// TIA Portal V19 export
ORGANIZATION_BLOCK "RT_Info_Cyclic"   // OB30, LAD, CyclicInterrupt
{ S7_Optimized_Access := 'TRUE' }
// stored: SetENOAutomatically false
   VAR_INPUT
      Initial_Call : Bool;   // Initial call of this OB
      Event_Count : Int;   // Events discarded
   END_VAR
   VAR CONSTANT
      constRunSoloState : Int := 37;
      constRunRedundant : Int := 40;
   END_VAR
   VAR_TEMP   // added for the SCL form of the ladder/FBD networks
      _w1 : Bool;
      _w2 : Bool;
      _w3 : Bool;
      _w4 : Bool;
   END_VAR
BEGIN

REGION Network 1: RT_Info for specific OB
   // Used to find the specific runtime of an OB, change the OB number and see the INFO.
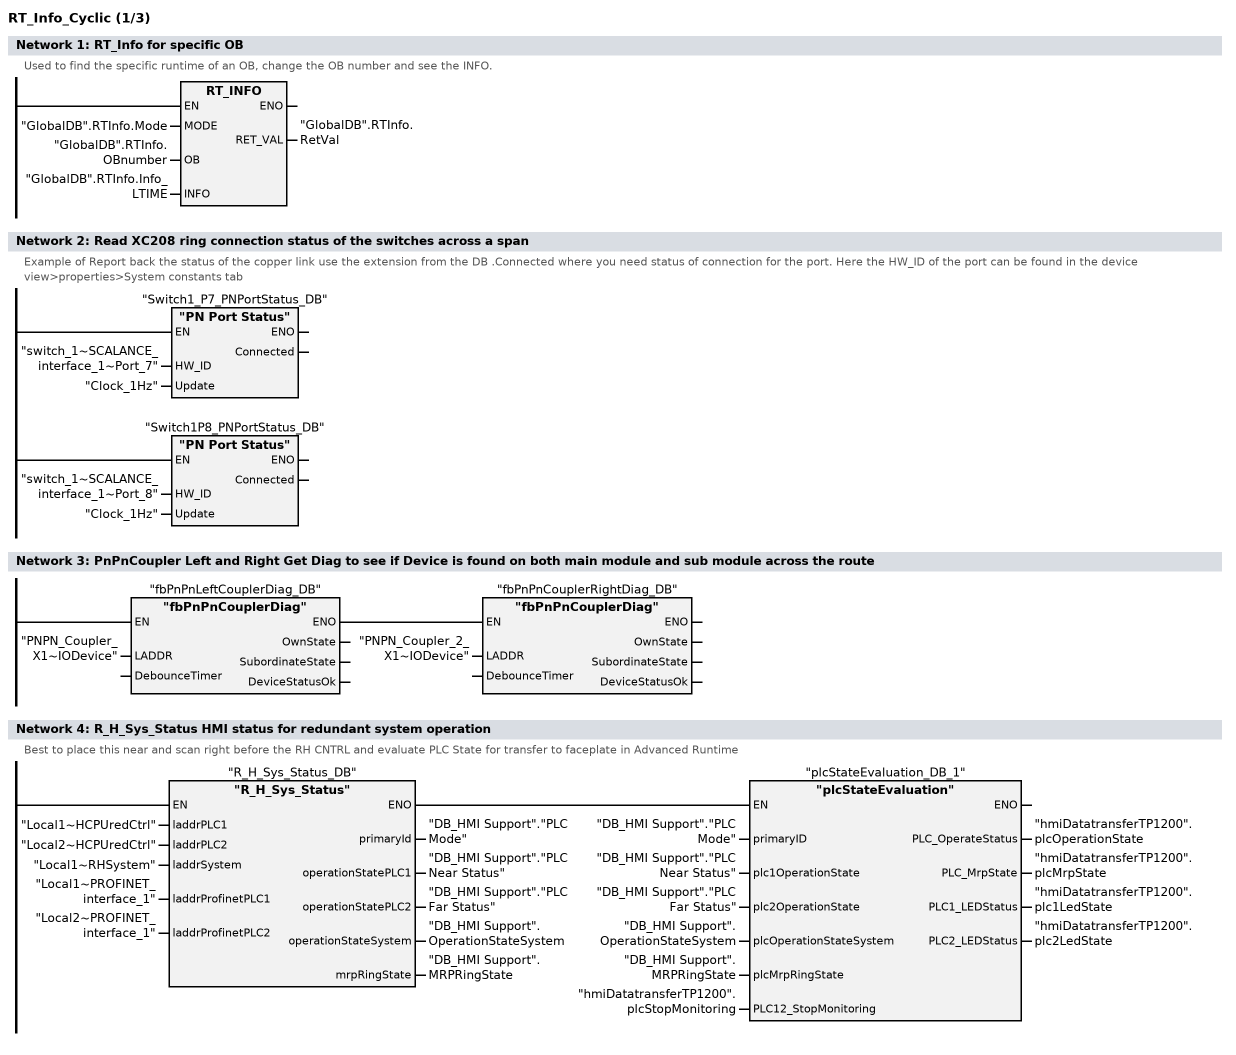
   RUNG wire#powerrail
      RT_INFO(MODE := "GlobalDB".RTInfo.Mode, OB := "GlobalDB".RTInfo.OBnumber, INFO := "GlobalDB".RTInfo.Info_LTIME, Ret_Val => "GlobalDB".RTInfo.RetVal)
   END_RUNG
   // the same network as SCL:
   "GlobalDB".RTInfo.RetVal := RT_INFO(MODE := "GlobalDB".RTInfo.Mode,
                           OB := "GlobalDB".RTInfo.OBnumber,
                           INFO := "GlobalDB".RTInfo.Info_LTIME);
END_REGION

REGION Network 2: Read XC208 ring connection status of the switches across a span
   // Example of Report back the status of the copper link use the extension from the DB .Connected where you need status of connection for the port. Here the HW_ID of the port can be found in the device view>properties>System constants tab
   RUNG wire#powerrail
      "Switch1_P7_PNPortStatus_DB"(HW_ID := "switch_1~SCALANCE_interface_1~Port_7", Update := "Clock_1Hz", Connected =>)
   END_RUNG
   RUNG wire#powerrail
      "Switch1P8_PNPortStatus_DB"(HW_ID := "switch_1~SCALANCE_interface_1~Port_8", Update := "Clock_1Hz", Connected =>)
   END_RUNG
   // the same network as SCL:
   "Switch1_P7_PNPortStatus_DB"(HW_ID := "switch_1~SCALANCE_interface_1~Port_7", Update := "Clock_1Hz");   // "PN Port Status"
   "Switch1P8_PNPortStatus_DB"(HW_ID := "switch_1~SCALANCE_interface_1~Port_8", Update := "Clock_1Hz");   // "PN Port Status"
END_REGION

REGION Network 3: PnPnCoupler Left and Right Get Diag to see if Device is found on both main module and sub module across the route
   RUNG wire#powerrail
      "fbPnPnLeftCouplerDiag_DB"(LADDR := "PNPN_Coupler_X1~IODevice", DebounceTimer :=, OwnState =>, SubordinateState =>, DeviceStatusOk =>)
      "fbPnPnCouplerRightDiag_DB"(LADDR := "PNPN_Coupler_2_X1~IODevice", DebounceTimer :=, OwnState =>, SubordinateState =>, DeviceStatusOk =>)
   END_RUNG
   // the same network as SCL:
   "fbPnPnLeftCouplerDiag_DB"(LADDR := "PNPN_Coupler_X1~IODevice", ENO => #_w1);   // "fbPnPnCouplerDiag"
   IF #_w1 THEN
       "fbPnPnCouplerRightDiag_DB"(LADDR := "PNPN_Coupler_2_X1~IODevice");   // "fbPnPnCouplerDiag"
   END_IF;
END_REGION

REGION Network 4: R_H_Sys_Status HMI status for redundant system operation
   // Best to place this near and scan right before the RH CNTRL and evaluate PLC State for transfer to faceplate in Advanced Runtime
   RUNG wire#powerrail
      "R_H_Sys_Status_DB"(laddrPLC1 := "Local1~HCPUredCtrl", laddrPLC2 := "Local2~HCPUredCtrl", laddrSystem := "Local1~RHSystem", laddrProfinetPLC1 := "Local1~PROFINET_interface_1", laddrProfinetPLC2 := "Local2~PROFINET_interface_1", primaryId => "DB_HMI Support"."PLC Mode", operationStatePLC1 => "DB_HMI Support"."PLC Near Status", operationStatePLC2 => "DB_HMI Support"."PLC Far Status", operationStateSystem => "DB_HMI Support".OperationStateSystem, mrpRingState => "DB_HMI Support".MRPRingState)
      "plcStateEvaluation_DB_1"(primaryID := "DB_HMI Support"."PLC Mode", plc1OperationState := "DB_HMI Support"."PLC Near Status", plc2OperationState := "DB_HMI Support"."PLC Far Status", plcOperationStateSystem := "DB_HMI Support".OperationStateSystem, plcMrpRingState := "DB_HMI Support".MRPRingState, PLC12_StopMonitoring := "hmiDatatransferTP1200".plcStopMonitoring, PLC_OperateStatus => "hmiDatatransferTP1200".plcOperationState, PLC_MrpState => "hmiDatatransferTP1200".plcMrpState, PLC1_LEDStatus => "hmiDatatransferTP1200".plc1LedState, PLC2_LEDStatus => "hmiDatatransferTP1200".plc2LedState)
   END_RUNG
   // the same network as SCL:
   "R_H_Sys_Status_DB"(laddrPLC1 := "Local1~HCPUredCtrl",   // "R_H_Sys_Status"
                       laddrPLC2 := "Local2~HCPUredCtrl",
                       laddrSystem := "Local1~RHSystem",
                       laddrProfinetPLC1 := "Local1~PROFINET_interface_1",
                       laddrProfinetPLC2 := "Local2~PROFINET_interface_1",
                       primaryId => "DB_HMI Support"."PLC Mode",
                       operationStatePLC1 => "DB_HMI Support"."PLC Near Status",
                       operationStatePLC2 => "DB_HMI Support"."PLC Far Status",
                       operationStateSystem => "DB_HMI Support".OperationStateSystem,
                       mrpRingState => "DB_HMI Support".MRPRingState,
                       ENO => #_w1);
   IF #_w1 THEN
       "plcStateEvaluation_DB_1"(primaryID := "DB_HMI Support"."PLC Mode",   // "plcStateEvaluation"
                               plc1OperationState := "DB_HMI Support"."PLC Near Status",
                               plc2OperationState := "DB_HMI Support"."PLC Far Status",
                               plcOperationStateSystem := "DB_HMI Support".OperationStateSystem,
                               plcMrpRingState := "DB_HMI Support".MRPRingState,
                               PLC12_StopMonitoring := "hmiDatatransferTP1200".plcStopMonitoring,
                               PLC_OperateStatus => "hmiDatatransferTP1200".plcOperationState,
                               PLC_MrpState => "hmiDatatransferTP1200".plcMrpState,
                               PLC1_LEDStatus => "hmiDatatransferTP1200".plc1LedState,
                               PLC2_LEDStatus => "hmiDatatransferTP1200".plc2LedState);
   END_IF;
END_REGION

REGION Network 5: Trigger primary stop RH_CNTRL
   // Self Latching Sequence using FullSwap Sequence tag, independent function with REQ tag
   // Used to trigger Primary Stop based on input from stop primary and full swap boolean tag;
   //  positive edge triggered instruction RH_CTRL below.
   // This network uses a Primary stop request, and evaluates if the RH_CTRL is busy before 
   // changing the mode or moving on to the next step.
   // The Retry_Busy tag is used to record if a Busy bit was in place while being triggered to prevent moving
   //  mode during middle of RH_CTRL operation.
   // 
   // Modes:
   // 3: Disable execution of the SYNCUP
   // 4: Re-enable execution of the SYNCUP
   // 7: Request SYNCUP system state 
   // 8: Request STOP of the primary CPU
   // 9: Request STOP of the backup CPU
   // 
   // Use mode 8 to stop the primary PLC, then use Mode 7 to Synch the primary and backup.
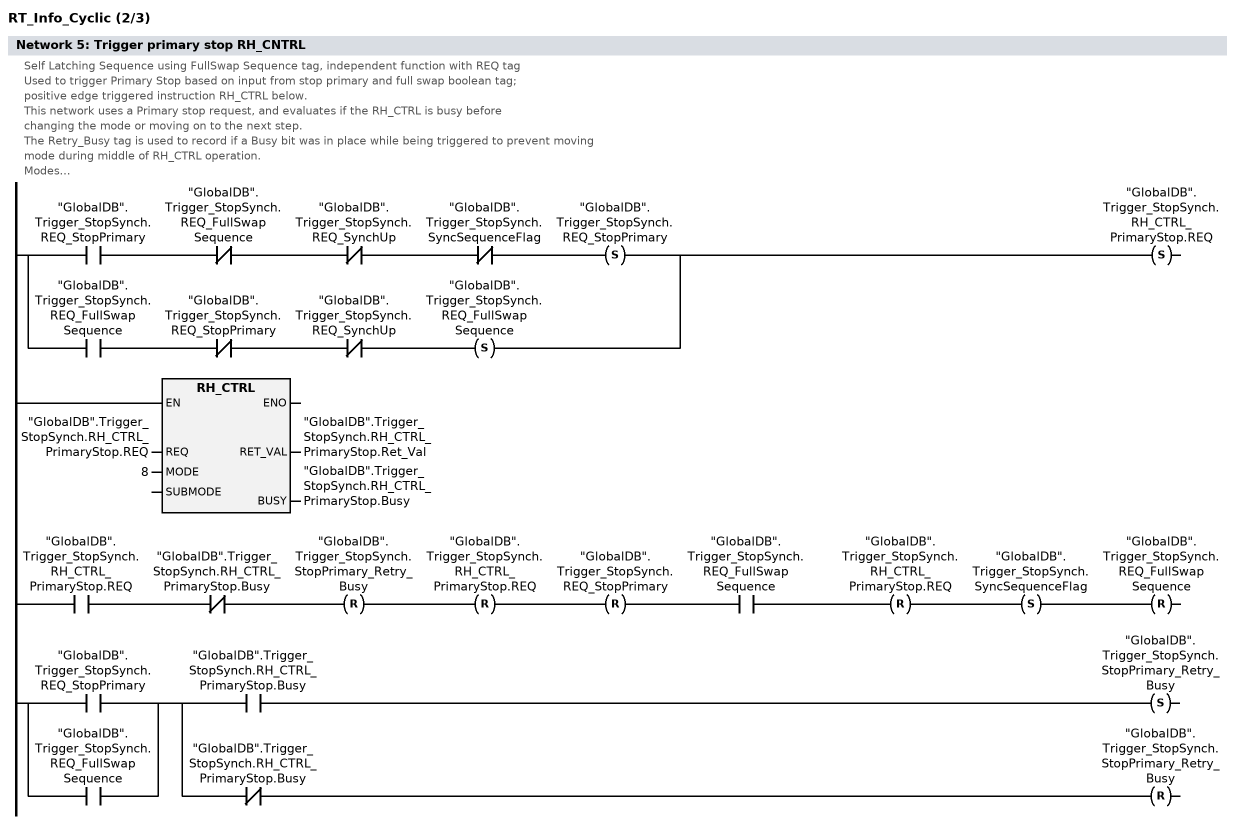
   RUNG wire#powerrail
      Contact( "GlobalDB".Trigger_StopSynch.REQ_StopPrimary )
      I_Contact( "GlobalDB".Trigger_StopSynch.REQ_FullSwapSequence )
      I_Contact( "GlobalDB".Trigger_StopSynch.REQ_SynchUp )
      I_Contact( "GlobalDB".Trigger_StopSynch.SyncSequenceFlag )
      S_Coil( "GlobalDB".Trigger_StopSynch.REQ_StopPrimary )
      wire#w1
      S_Coil( "GlobalDB".Trigger_StopSynch.RH_CTRL_PrimaryStop.REQ )
   END_RUNG
   RUNG wire#powerrail
      Contact( "GlobalDB".Trigger_StopSynch.REQ_FullSwapSequence )
      I_Contact( "GlobalDB".Trigger_StopSynch.REQ_StopPrimary )
      I_Contact( "GlobalDB".Trigger_StopSynch.REQ_SynchUp )
      S_Coil( "GlobalDB".Trigger_StopSynch.REQ_FullSwapSequence )
   END_RUNG wire#w1
   RUNG wire#powerrail
      RH_CTRL(REQ := "GlobalDB".Trigger_StopSynch.RH_CTRL_PrimaryStop.REQ, Mode := 8, Submode :=, Ret_Val => "GlobalDB".Trigger_StopSynch.RH_CTRL_PrimaryStop.Ret_Val, Busy => "GlobalDB".Trigger_StopSynch.RH_CTRL_PrimaryStop.Busy)
   END_RUNG
   RUNG wire#powerrail
      Contact( "GlobalDB".Trigger_StopSynch.RH_CTRL_PrimaryStop.REQ )
      I_Contact( "GlobalDB".Trigger_StopSynch.RH_CTRL_PrimaryStop.Busy )
      R_Coil( "GlobalDB".Trigger_StopSynch.StopPrimary_Retry_Busy )
      R_Coil( "GlobalDB".Trigger_StopSynch.RH_CTRL_PrimaryStop.REQ )
      R_Coil( "GlobalDB".Trigger_StopSynch.REQ_StopPrimary )
      Contact( "GlobalDB".Trigger_StopSynch.REQ_FullSwapSequence )
      R_Coil( "GlobalDB".Trigger_StopSynch.RH_CTRL_PrimaryStop.REQ )
      S_Coil( "GlobalDB".Trigger_StopSynch.SyncSequenceFlag )
      R_Coil( "GlobalDB".Trigger_StopSynch.REQ_FullSwapSequence )
   END_RUNG
   RUNG wire#powerrail
      Contact( "GlobalDB".Trigger_StopSynch.REQ_StopPrimary )
      wire#w2
      Contact( "GlobalDB".Trigger_StopSynch.RH_CTRL_PrimaryStop.Busy )
      S_Coil( "GlobalDB".Trigger_StopSynch.StopPrimary_Retry_Busy )
   END_RUNG
   RUNG wire#powerrail
      Contact( "GlobalDB".Trigger_StopSynch.REQ_FullSwapSequence )
   END_RUNG wire#w2
   RUNG wire#w2
      I_Contact( "GlobalDB".Trigger_StopSynch.RH_CTRL_PrimaryStop.Busy )
      R_Coil( "GlobalDB".Trigger_StopSynch.StopPrimary_Retry_Busy )
   END_RUNG
   // the same network as SCL:
   #_w1 := "GlobalDB".Trigger_StopSynch.REQ_StopPrimary AND NOT "GlobalDB".Trigger_StopSynch.REQ_FullSwapSequence AND NOT "GlobalDB".Trigger_StopSynch.REQ_SynchUp AND NOT "GlobalDB".Trigger_StopSynch.SyncSequenceFlag;
   IF #_w1 THEN "GlobalDB".Trigger_StopSynch.REQ_StopPrimary := TRUE; END_IF;
   #_w2 := "GlobalDB".Trigger_StopSynch.REQ_FullSwapSequence AND NOT "GlobalDB".Trigger_StopSynch.REQ_StopPrimary AND NOT "GlobalDB".Trigger_StopSynch.REQ_SynchUp;
   IF #_w2 THEN "GlobalDB".Trigger_StopSynch.REQ_FullSwapSequence := TRUE; END_IF;
   IF #_w1 OR #_w2 THEN "GlobalDB".Trigger_StopSynch.RH_CTRL_PrimaryStop.REQ := TRUE; END_IF;
   "GlobalDB".Trigger_StopSynch.RH_CTRL_PrimaryStop.Ret_Val := RH_CTRL(REQ := "GlobalDB".Trigger_StopSynch.RH_CTRL_PrimaryStop.REQ,
                           Mode := 8,
                           Busy => "GlobalDB".Trigger_StopSynch.RH_CTRL_PrimaryStop.Busy);
   #_w3 := "GlobalDB".Trigger_StopSynch.RH_CTRL_PrimaryStop.REQ AND NOT "GlobalDB".Trigger_StopSynch.RH_CTRL_PrimaryStop.Busy;
   IF #_w3 THEN
       "GlobalDB".Trigger_StopSynch.StopPrimary_Retry_Busy := FALSE;
       "GlobalDB".Trigger_StopSynch.RH_CTRL_PrimaryStop.REQ := FALSE;
       "GlobalDB".Trigger_StopSynch.REQ_StopPrimary := FALSE;
   END_IF;
   IF #_w3 AND "GlobalDB".Trigger_StopSynch.REQ_FullSwapSequence THEN
       "GlobalDB".Trigger_StopSynch.RH_CTRL_PrimaryStop.REQ := FALSE;
       "GlobalDB".Trigger_StopSynch.SyncSequenceFlag := TRUE;
       "GlobalDB".Trigger_StopSynch.REQ_FullSwapSequence := FALSE;
   END_IF;
   #_w4 := "GlobalDB".Trigger_StopSynch.REQ_StopPrimary OR "GlobalDB".Trigger_StopSynch.REQ_FullSwapSequence;
   IF #_w4 AND "GlobalDB".Trigger_StopSynch.RH_CTRL_PrimaryStop.Busy THEN
       "GlobalDB".Trigger_StopSynch.StopPrimary_Retry_Busy := TRUE;
   END_IF;
   IF #_w4 AND NOT "GlobalDB".Trigger_StopSynch.RH_CTRL_PrimaryStop.Busy THEN
       "GlobalDB".Trigger_StopSynch.StopPrimary_Retry_Busy := FALSE;
   END_IF;
END_REGION

REGION Network 6: Trigger Synch up RH_CNTRL
   // Self Latching Sequence using FullSwap Sequence tag, independent function with REQ tag
   // Used to trigger Sync up; positive edge triggered instruction RH_CTRL below
   // Sequence can also be triggered by Full sequence request which can set the SyncSequenceFlag below
   // SyncSequence Flag is help for next step until run Run-Solo status is reported
   //  positive edge triggered instruction RH_CTRL below
   // This network uses a synch up request, and evaluates if the RH_CTRL is busy before changing the mode
   // The Retry_Busy tag is used to record if a Busy bit was in place while being triggered to prevent moving
   //  mode during middle of RH_CTRL operation
   // 
   // Modes:
   // 3: Disable execution of the SYNCUP
   // 4: Re-enable execution of the SYNCUP
   // 7: Request SYNCUP system state 
   // 8: Request STOP of the primary CPU
   // 9: Request STOP of the backup CPU
   // 
   // Use mode 8 to stop the primary PLC, then use Mode 7 to Synch the primary and backup.
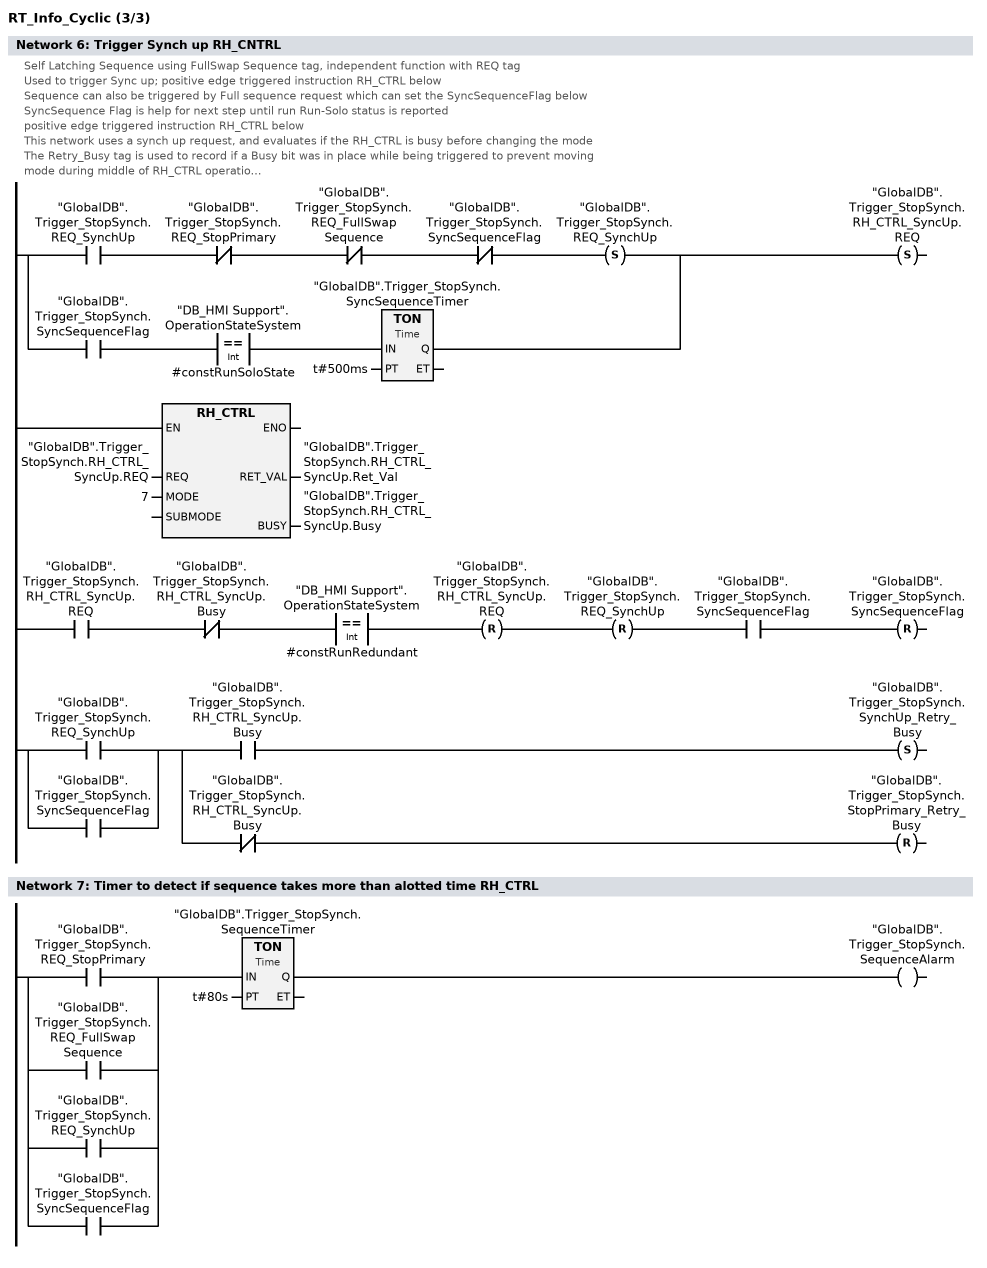
   RUNG wire#powerrail
      Contact( "GlobalDB".Trigger_StopSynch.REQ_SynchUp )
      I_Contact( "GlobalDB".Trigger_StopSynch.REQ_StopPrimary )
      I_Contact( "GlobalDB".Trigger_StopSynch.REQ_FullSwapSequence )
      I_Contact( "GlobalDB".Trigger_StopSynch.SyncSequenceFlag )
      S_Coil( "GlobalDB".Trigger_StopSynch.REQ_SynchUp )
      wire#w1
      S_Coil( "GlobalDB".Trigger_StopSynch.RH_CTRL_SyncUp.REQ )
   END_RUNG
   RUNG wire#powerrail
      Contact( "GlobalDB".Trigger_StopSynch.SyncSequenceFlag )
      { S7_Templates := "SrcType := Int" } EQ_Contact(in1 := "DB_HMI Support".OperationStateSystem, in2 := #constRunSoloState)
      { S7_Templates := "time_type := Time" } "GlobalDB".Trigger_StopSynch.SyncSequenceTimer.TON(pt := t#500ms, et =>)
   END_RUNG wire#w1
   RUNG wire#powerrail
      RH_CTRL(REQ := "GlobalDB".Trigger_StopSynch.RH_CTRL_SyncUp.REQ, Mode := 7, Submode :=, Ret_Val => "GlobalDB".Trigger_StopSynch.RH_CTRL_SyncUp.Ret_Val, Busy => "GlobalDB".Trigger_StopSynch.RH_CTRL_SyncUp.Busy)
   END_RUNG
   RUNG wire#powerrail
      Contact( "GlobalDB".Trigger_StopSynch.RH_CTRL_SyncUp.REQ )
      I_Contact( "GlobalDB".Trigger_StopSynch.RH_CTRL_SyncUp.Busy )
      { S7_Templates := "SrcType := Int" } EQ_Contact(in1 := "DB_HMI Support".OperationStateSystem, in2 := #constRunRedundant)
      R_Coil( "GlobalDB".Trigger_StopSynch.RH_CTRL_SyncUp.REQ )
      R_Coil( "GlobalDB".Trigger_StopSynch.REQ_SynchUp )
      Contact( "GlobalDB".Trigger_StopSynch.SyncSequenceFlag )
      R_Coil( "GlobalDB".Trigger_StopSynch.SyncSequenceFlag )
   END_RUNG
   RUNG wire#powerrail
      Contact( "GlobalDB".Trigger_StopSynch.REQ_SynchUp )
      wire#w2
      Contact( "GlobalDB".Trigger_StopSynch.RH_CTRL_SyncUp.Busy )
      S_Coil( "GlobalDB".Trigger_StopSynch.SynchUp_Retry_Busy )
   END_RUNG
   RUNG wire#powerrail
      Contact( "GlobalDB".Trigger_StopSynch.SyncSequenceFlag )
   END_RUNG wire#w2
   RUNG wire#w2
      I_Contact( "GlobalDB".Trigger_StopSynch.RH_CTRL_SyncUp.Busy )
      R_Coil( "GlobalDB".Trigger_StopSynch.StopPrimary_Retry_Busy )
   END_RUNG
   // the same network as SCL:
   #_w1 := "GlobalDB".Trigger_StopSynch.REQ_SynchUp AND NOT "GlobalDB".Trigger_StopSynch.REQ_StopPrimary AND NOT "GlobalDB".Trigger_StopSynch.REQ_FullSwapSequence AND NOT "GlobalDB".Trigger_StopSynch.SyncSequenceFlag;
   IF #_w1 THEN "GlobalDB".Trigger_StopSynch.REQ_SynchUp := TRUE; END_IF;
   "GlobalDB".Trigger_StopSynch.SyncSequenceTimer.TON(IN := "GlobalDB".Trigger_StopSynch.SyncSequenceFlag AND ("DB_HMI Support".OperationStateSystem = #constRunSoloState),
                           PT := t#500ms);
   IF #_w1 OR "GlobalDB".Trigger_StopSynch.SyncSequenceTimer.Q THEN
       "GlobalDB".Trigger_StopSynch.RH_CTRL_SyncUp.REQ := TRUE;
   END_IF;
   "GlobalDB".Trigger_StopSynch.RH_CTRL_SyncUp.Ret_Val := RH_CTRL(REQ := "GlobalDB".Trigger_StopSynch.RH_CTRL_SyncUp.REQ,
                           Mode := 7,
                           Busy => "GlobalDB".Trigger_StopSynch.RH_CTRL_SyncUp.Busy);
   #_w2 := "GlobalDB".Trigger_StopSynch.RH_CTRL_SyncUp.REQ AND NOT "GlobalDB".Trigger_StopSynch.RH_CTRL_SyncUp.Busy AND ("DB_HMI Support".OperationStateSystem = #constRunRedundant);
   IF #_w2 THEN
       "GlobalDB".Trigger_StopSynch.RH_CTRL_SyncUp.REQ := FALSE;
       "GlobalDB".Trigger_StopSynch.REQ_SynchUp := FALSE;
   END_IF;
   IF #_w2 AND "GlobalDB".Trigger_StopSynch.SyncSequenceFlag THEN
       "GlobalDB".Trigger_StopSynch.SyncSequenceFlag := FALSE;
   END_IF;
   #_w3 := "GlobalDB".Trigger_StopSynch.REQ_SynchUp OR "GlobalDB".Trigger_StopSynch.SyncSequenceFlag;
   IF #_w3 AND "GlobalDB".Trigger_StopSynch.RH_CTRL_SyncUp.Busy THEN
       "GlobalDB".Trigger_StopSynch.SynchUp_Retry_Busy := TRUE;
   END_IF;
   IF #_w3 AND NOT "GlobalDB".Trigger_StopSynch.RH_CTRL_SyncUp.Busy THEN
       "GlobalDB".Trigger_StopSynch.StopPrimary_Retry_Busy := FALSE;
   END_IF;
END_REGION

REGION Network 7: Timer to detect if sequence takes more than alotted time RH_CTRL
   RUNG wire#powerrail
      Contact( "GlobalDB".Trigger_StopSynch.REQ_StopPrimary )
      wire#w1
      { S7_Templates := "time_type := Time" } "GlobalDB".Trigger_StopSynch.SequenceTimer.TON(pt := t#80s, et =>)
      Coil( "GlobalDB".Trigger_StopSynch.SequenceAlarm )
   END_RUNG
   RUNG wire#powerrail
      Contact( "GlobalDB".Trigger_StopSynch.REQ_FullSwapSequence )
   END_RUNG wire#w1
   RUNG wire#powerrail
      Contact( "GlobalDB".Trigger_StopSynch.REQ_SynchUp )
   END_RUNG wire#w1
   RUNG wire#powerrail
      Contact( "GlobalDB".Trigger_StopSynch.SyncSequenceFlag )
   END_RUNG wire#w1
   // the same network as SCL:
   "GlobalDB".Trigger_StopSynch.SequenceTimer.TON(IN := "GlobalDB".Trigger_StopSynch.REQ_StopPrimary OR "GlobalDB".Trigger_StopSynch.REQ_FullSwapSequence OR "GlobalDB".Trigger_StopSynch.REQ_SynchUp OR "GlobalDB".Trigger_StopSynch.SyncSequenceFlag,
                           PT := t#80s);
   "GlobalDB".Trigger_StopSynch.SequenceAlarm := "GlobalDB".Trigger_StopSynch.SequenceTimer.Q;
END_REGION
END_ORGANIZATION_BLOCK
